// Mitsubishi GX Developer project: single   PLC: FX3U

PROGRAM MAIN
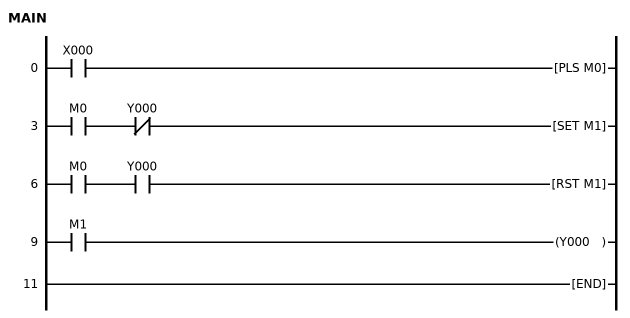
0     LD      X000
      PLS     M0
3     LD      M0
      ANI     Y000
      SET     M1
6     LD      M0
      AND     Y000
      RST     M1
9     LD      M1
      OUT     Y000
11    END
END_PROGRAM
